// TIA Portal V20 export
TYPE "LER_typeIntlockAll"
// stored: Access Published
   STRUCT
      Actuator { S7_SetPoint := 'True'} : "LER_typeAxisActuatorCondition";
      Home { S7_SetPoint := 'True'} : "LER_typeAxisHomeCondition";
      Jog { S7_SetPoint := 'True'} : "LER_typeAxisJogCondition";
      Position { S7_SetPoint := 'True'} : "LER_typeAxisPositionCondition";
   END_STRUCT;
END_TYPE
